# EPICS autosave request: apps/iocBoot/ioclakeshore450/lakeshore_settings.req
file lakeshore450_settings.req P=HPS:,R=LS450_1:
file lakeshore450_settings.req P=HPS:,R=LS450_2:
